PROGRAM Runtime_Control
VAR
	RuntimeActivate: BOOL;
	FRA3RT: Production_Runtime_Values;
	BackupCanCounterA: CTU;
	BackCanCounterA_CurrentCount: WORD;
	ResetBackupCounterA: BOOL;
	BackupCanCounterB: CTU;
	BackCanCounterB_CurrentCount: WORD;
	MultiplierValue_FOR_BackupCounterB: DINT;

	FRA3_Downtime_LOG: FB_Downtime_LOG;
	DowntimeDetected: BOOL;
	ResetStopReasonsValues: F_TRIG;
END_VAR

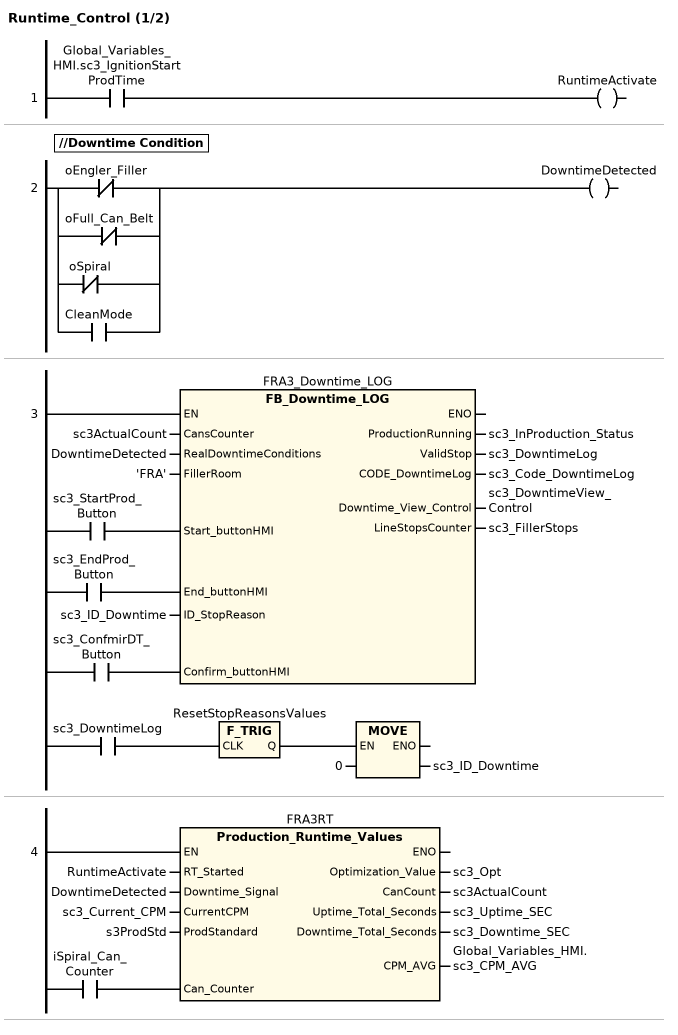
// NETWORK 1
RuntimeActivate := Global_Variables_HMI.sc3_IgnitionStartProdTime;

// NETWORK 2
// label: //Downtime Condition
DowntimeDetected := NOT oEngler_Filler OR NOT oFull_Can_Belt OR NOT oSpiral OR CleanMode;

// NETWORK 3
FRA3_Downtime_LOG(
    CansCounter := sc3ActualCount,
    RealDowntimeConditions := DowntimeDetected,
    FillerRoom := 'FRA',
    Start_buttonHMI := sc3_StartProd_Button,
    End_buttonHMI := sc3_EndProd_Button,
    ID_StopReason := sc3_ID_Downtime,
    Confirm_buttonHMI := sc3_ConfmirDT_Button,
    ProductionRunning => sc3_InProduction_Status,
    ValidStop => sc3_DowntimeLog,
    CODE_DowntimeLog => sc3_Code_DowntimeLog,
    Downtime_View_Control => sc3_DowntimeView_Control,
    LineStopsCounter => sc3_FillerStops); // FB_Downtime_LOG
ResetStopReasonsValues(CLK := sc3_DowntimeLog); // F_TRIG
IF ResetStopReasonsValues.Q THEN sc3_ID_Downtime := 0; END_IF

// NETWORK 4
FRA3RT(
    RT_Started := RuntimeActivate,
    Downtime_Signal := DowntimeDetected,
    CurrentCPM := sc3_Current_CPM,
    ProdStandard := s3ProdStd,
    Can_Counter := iSpiral_Can_Counter,
    Optimization_Value => sc3_Opt,
    CanCount => sc3ActualCount,
    Uptime_Total_Seconds => sc3_Uptime_SEC,
    Downtime_Total_Seconds => sc3_Downtime_SEC,
    CPM_AVG => Global_Variables_HMI.sc3_CPM_AVG); // Production_Runtime_Values

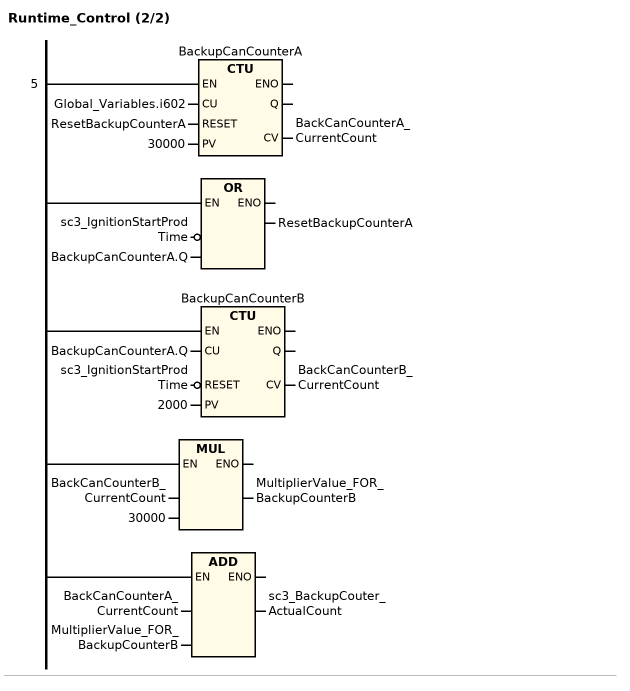
// NETWORK 5
BackupCanCounterA(
    CU := Global_Variables.i602,
    RESET := ResetBackupCounterA,
    PV := 30000,
    CV => BackCanCounterA_CurrentCount); // CTU
ResetBackupCounterA := NOT sc3_IgnitionStartProdTime OR BackupCanCounterA.Q;
BackupCanCounterB(
    CU := BackupCanCounterA.Q,
    RESET := NOT sc3_IgnitionStartProdTime,
    PV := 2000,
    CV => BackCanCounterB_CurrentCount); // CTU
MultiplierValue_FOR_BackupCounterB := BackCanCounterB_CurrentCount * 30000;
sc3_BackupCouter_ActualCount := BackCanCounterA_CurrentCount + MultiplierValue_FOR_BackupCounterB;

END_PROGRAM

(* stored: Version 1.1.0.1, ProductVersion 3.1.4024.15
   POU Runtime_Control: Id {cfb32c9e-88d0-42c6-9b77-e1441cd66f93}, SpecialFunc None *)
